Universal Robots PolyScope program: DMT08b_6.urp

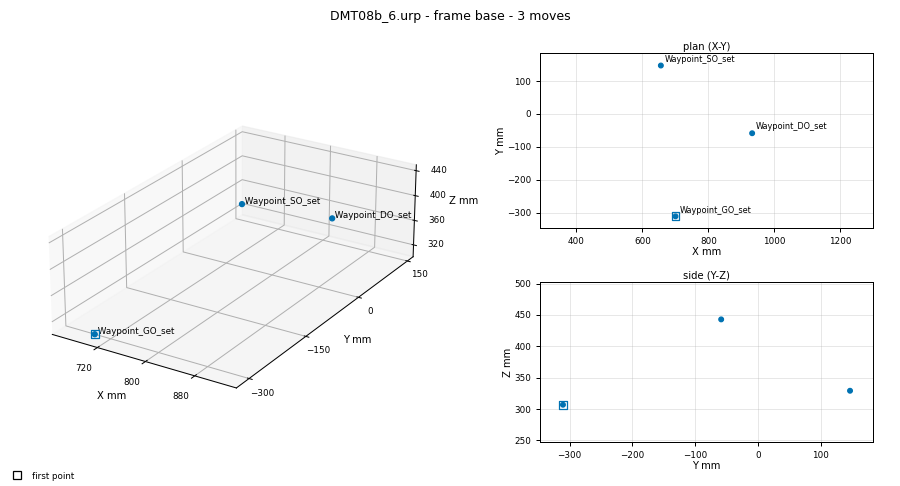
[picture p0: tool path of DMT08b_6.urp in frame base, 3 of 13 moves have a stored position in this frame; points joined in program order, loops and branches not executed]
Program DMT08b_6 (installation=default directory=/programs/usbdisk createdIn=3.5.0.10584 lastSavedIn=3.15.8.106339 robotSerialNumber=2017307354)
Calibrated DH parameters: a=[-0.000055, -0.610354, -0.571266, 0.000097, 0.000056, 0]; d=[0.128196, 3.8936, -4.338276, 0.608123, 0.115639, 0.092138]; alpha=[1.57086, -0.013529, -0.012604, 1.570975, -1.570813, 0]; deltaTheta=[-0.000051, -0.086091, 0.095923, -0.009846, -0.000078, 0.000069]
BeforeStart
  Script: enable_external_ft_sensor( True , sensor_mass = 0.0,  sensor_measuring_offset = [0.0, 0.0, 0.0], sensor_cog = [0.0, 0.0, 0.0] )
  sock_res := True
  Loop While (checkContinuously=false) expression=not sock_res
    Script: sock_res=socket_open("192.168.1.30",1000)
  res := ""
  Loop While (checkContinuously=false) expression=res ≟ ""
    Script: socket_send_line("TARE(1)")
    Script: res=socket_read_string()
  Script: write_output_boolean_register(0, False)
  Wait Sleep waitTime=0.01
  Script: popup("Registers reset, run PC code and then click Continue", title="Hi DMT", blocking = True)
  mode := 0
Robot Program (runOnlyOnce=true)
  Script: write_output_boolean_register(0, True)
  Script: sync()
  Loop While (checkContinuously=false) expression=mode<4
    Loop While (checkContinuously=true) expression=mode==1
      Script: write_output_boolean_register(0, True)
      Script: sync()
      MoveL speed 250 mm/s, acceleration 1200 mm/s^2 (useActiveTCP=true) feature=Base
        Waypoint Waypoint_GO_set: TCP in base x=700.482 y=-310.573 z=306.908 mm, rx=3.141 ry=0.0001 rz=-0.0001 rad; joints [143.166, -74.81, 109.164, -124.372, 269.248, 233.493] deg
      SuppressedNode
        Force Simple feature=Base; selection=[0, 0, 1, 0, 0, 0]; wrench=[0, 0, -20, 0, 0, 0]; limitsForce=[0.15, 0.15, 0.15, 1.047198, 1.047198, 1.047198]; limitsMotion=[0.1, 0.1, 0.1, 0.349066, 0.349066, 0.349066]
          Wait Sleep waitTime=0.5
      MoveL speed 150 mm/s, acceleration 2225 mm/s^2 (useActiveTCP=false) feature=Base
        Waypoint Waypoint_G12 (Relative): relativeFromPosition TCP in base x=504.862 y=-222.419 z=97.846 mm, rx=3.141 ry=0 rz=0 rad; joints [144.817, -64.31, 112.427, -138.137, 269.972, 234.817] deg; TCP in base x=409.862 y=-222.419 z=97.846 mm, rx=3.141 ry=0 rz=0 rad; joints [137.981, -72.866, 126.336, -143.492, 269.975, 227.981] deg
      Loop Counting (count=4) loopVariable(name=Loop_8)
        MoveL speed 50 mm/s, acceleration 300 mm/s^2 (useActiveTCP=true) feature=Base
          Waypoint Waypoint_G23 (Relative): relativeFromPosition TCP in base x=409.862 y=-222.419 z=97.846 mm, rx=3.141 ry=0 rz=0 rad; joints [137.981, -72.866, 126.336, -143.492, 269.975, 227.981] deg; TCP in base x=409.862 y=-222.419 z=100.846 mm, rx=3.141 ry=0 rz=0 rad; joints [137.981, -73.268, 126.217, -142.972, 269.975, 227.981] deg
        MoveL speed 100 mm/s, acceleration 200 mm/s^2 (useActiveTCP=false) feature=Base
          Waypoint Waypoint_G34 (Relative): relativeFromPosition TCP in base x=409.862 y=-222.419 z=98.846 mm, rx=3.141 ry=0 rz=0 rad; joints [137.981, -73, 126.297, -143.319, 269.975, 227.981] deg; TCP in base x=504.862 y=-177.419 z=98.846 mm, rx=3.141 ry=0 rz=0 rad; joints [148.873, -66.067, 115.171, -139.121, 269.971, 238.873] deg
        MoveL speed 50 mm/s, acceleration 300 mm/s^2 (useActiveTCP=true) feature=Base
          Waypoint Waypoint_G4O (Relative): relativeFromPosition TCP in base x=409.862 y=-222.419 z=100.846 mm, rx=3.141 ry=0 rz=0 rad; joints [137.981, -73.268, 126.217, -142.972, 269.975, 227.981] deg; TCP in base x=409.862 y=-222.419 z=98.846 mm, rx=3.141 ry=0 rz=0 rad; joints [137.981, -73, 126.297, -143.319, 269.975, 227.981] deg
        SuppressedNode
          Force Simple feature=Base; selection=[0, 0, 1, 0, 0, 0]; wrench=[0, 0, -20, 0, 0, 0]; limitsForce=[0.15, 0.15, 0.15, 1.047198, 1.047198, 1.047198]; limitsMotion=[0.1, 0.1, 0.1, 0.349066, 0.349066, 0.349066]
            Wait Sleep waitTime=0.5
        MoveL speed 150 mm/s, acceleration 2225 mm/s^2 (useActiveTCP=false) feature=Base
          Waypoint Waypoint_G12 (Relative): relativeFromPosition TCP in base x=504.862 y=-222.419 z=97.846 mm, rx=3.141 ry=0 rz=0 rad; joints [144.817, -64.31, 112.427, -138.137, 269.972, 234.817] deg; TCP in base x=409.862 y=-222.419 z=97.846 mm, rx=3.141 ry=0 rz=0 rad; joints [137.981, -72.866, 126.336, -143.492, 269.975, 227.981] deg
      Script: write_output_boolean_register(0, False)
      Script: sync()
    Loop While (checkContinuously=true) expression=mode==2
      Script: write_output_boolean_register(0, True)
      Script: write_output_boolean_register(32, True)
      Script: sync()
      Wait Sleep waitTime=0.5
      MoveL speed 250 mm/s, acceleration 1200 mm/s^2 (useActiveTCP=true) feature=Base
        Waypoint Waypoint_DO_set: TCP in base x=932.962 y=-58.379 z=442.977 mm, rx=3.141 ry=0.0001 rz=0.0001 rad; joints [165.794, -65.483, 81.029, -105.558, 269.02, 256.304] deg
        Waypoint Waypoint_DO1 (Relative): relativeFromPosition TCP in base x=658.55 y=-49.546 z=529.242 mm, rx=3.1409 ry=0.0002 rz=0 rad; joints [166.189, -63.237, 41.872, -68.645, 269.959, 256.184] deg; TCP in base x=658.55 y=-49.546 z=499.242 mm, rx=3.1409 ry=0.0002 rz=0 rad; joints [166.189, -65.044, 49.207, -74.172, 269.959, 256.184] deg
      Script: write_output_boolean_register(32, False)
      Wait Sleep waitTime=1
      MoveL speed 250 mm/s, acceleration 1200 mm/s^2 (useActiveTCP=true) feature=Base
        Waypoint Waypoint_D1O (Relative): relativeFromPosition TCP in base x=658.55 y=-49.546 z=499.242 mm, rx=3.1409 ry=0.0002 rz=0 rad; joints [166.189, -65.044, 49.207, -74.172, 269.959, 256.184] deg; TCP in base x=658.55 y=-49.546 z=529.242 mm, rx=3.1409 ry=0.0002 rz=0 rad; joints [166.189, -63.237, 41.872, -68.645, 269.959, 256.184] deg
      Script: write_output_boolean_register(0, False)
      Script: sync()
    Loop While (checkContinuously=true) expression=mode==3
      Script: write_output_boolean_register(0, True)
      Script: write_output_boolean_register(32, True)
      Script: sync()
      MoveL speed 100 mm/s, acceleration 200 mm/s^2 (useActiveTCP=false) feature=Base
        Waypoint Waypoint_SO_set: TCP in base x=656.036 y=147.031 z=329.213 mm, rx=3.141 ry=0 rz=-0.0002 rad; joints [177.912, -84.28, 118.105, -123.82, 269.368, 268.263] deg
      Script: write_output_boolean_register(32, False)
      Script: sync()
      MoveL speed 100 mm/s, acceleration 200 mm/s^2 (useActiveTCP=true) feature=Base
        Waypoint Waypoint_SO1 (Relative): relativeFromPosition TCP in base x=432.881 y=108.144 z=221.86 mm, rx=3.141 ry=0 rz=0 rad; joints [179.873, -89.103, 121.463, -122.36, 269.966, 269.873] deg; TCP in base x=522.881 y=108.144 z=221.86 mm, rx=3.141 ry=0 rz=0 rad; joints [179.895, -77.675, 108.365, -120.69, 269.966, 269.895] deg
      Script: write_output_boolean_register(32, True)
      Script: sync()
      MoveL speed 100 mm/s, acceleration 200 mm/s^2 (useActiveTCP=true) feature=Base
        Waypoint Waypoint_S12 (Relative): relativeFromPosition TCP in base x=522.881 y=108.144 z=221.86 mm, rx=3.141 ry=0 rz=0 rad; joints [179.895, -77.675, 108.365, -120.69, 269.966, 269.895] deg; TCP in base x=482.88 y=108.144 z=181.86 mm, rx=3.141 ry=0 rz=0 rad; joints [179.886, -79.194, 117.374, -128.18, 269.966, 269.886] deg
      Force Simple feature=Base; selection=[0, 0, 1, 0, 0, 0]; wrench=[0, 0, -6, 0, 0, 0]; limitsForce=[0.15, 0.15, 0.15, 1.047198, 1.047198, 1.047198]; limitsMotion=[0.1, 0.1, 0.1, 0.349066, 0.349066, 0.349066]
        Wait Sleep waitTime=0.5
        Script: write_output_boolean_register(32, False)
        Script: sync()
        MoveL speed 30 mm/s, acceleration 200 mm/s^2 (useActiveTCP=false) feature=Base
          Waypoint Waypoint_S23 (Relative): relativeFromPosition TCP in base x=492.777 y=108.199 z=182.69 mm, rx=3.141 ry=0 rz=0 rad; joints [179.895, -78.093, 115.821, -127.728, 269.966, 269.895] deg; TCP in base x=402.777 y=108.199 z=182.69 mm, rx=3.141 ry=0 rz=0 rad; joints [179.872, -89.337, 128.769, -129.432, 269.966, 269.872] deg
        Script: write_output_boolean_register(32, True)
        Script: sync()
      Script: write_output_boolean_register(0, False)
      Script: sync()
    Loop While (checkContinuously=true) expression=mode==4
      Halt
  Script: sync()
Thread Thread_1 (runOnlyOnce=false)
  tmp := p[0,0,0,0,0,0]
  Loop Forever
    Script file /home/ur/ursim/ursim-3.15.0.106151/programs/pose_register.script
      | tmp[0]=read_input_float_register(0)
      | tmp[1]=read_input_float_register(1)
      | tmp[2]=read_input_float_register(2)
      | tmp[3]=read_input_float_register(3)
      | tmp[4]=read_input_float_register(4)
      | tmp[5]=read_input_float_register(5)
    Script: sync()
    mode := read_input_integer_register(0)
    Script: sync()
